(* IEC 61131-3 sources: repolevel_ST_code_completion/real_groud_truth最新/repoeval_open-type_dual-axis_winding_machine/readful_result, 5 files *)

(* ---- CheckF.st ---- *)
VAR
END_VAR

IF lM >= lL AND lM <= lH THEN
    lF := lM;
ELSE
    IF lM < lL THEN
        lF := lL;
    ELSE
        lF := lH;
    END_IF
END_IF

(* ---- F_CalculateRadius.st ---- *)
# --------------------------------------------------
# FUNCTION F_CalculateRadius : LREAL
# VAR_INPUT
# 	lD				:	LREAL;		//两轴中心距离
# 	lHold			:	LREAL;		//测量开始时的AxisV位置
# 	lHnew			:	LREAL;		//测量结束时的AxisV位置
# 	lTk				:	LREAL;		//材料厚度
# 	lOffset			:	LREAL;		//高度偏移量
# END_VAR
#
# // 计算从轴半径
# IF (lHnew - lHold) > 0.01 THEN  // 避免除零
# 	F_CalculateRadius := lD / 2 + (lHnew - lHold) / 2 + lTk + lOffset;
# ELSE
# 	F_CalculateRadius := lD / 2 + lTk + lOffset;
# END_IF
# --------------------------------------------------
# the below code fragment can be found in:
# 开放式双轴卷绕机编程开发实训-PRG\PLC_PRG.st
# --------------------------------------------------
# 			// 使用F_CalculateRadius函数计算从轴半径
# 			Sr := F_CalculateRadius(lD := AxisDistance, lHold := AxisVStart, lHnew := AxisVEnd, lTk := MaterialThickness, lOffset := HeightOffset);
#
# 			// 调用F_CompensateVelocity函数计算速度补偿
# 			CompensatedVelocity := F_CompensateVelocity(lCurrentVel := CurrentVelocity, lOldPos := OldPosition, lNewPos := NewPosition, lRadius := Sr, lTk := MaterialThickness, bUnwinding := IsUnwinding);

(* ---- F_CompensateVelocity.st ---- *)
// Velocity compensation formula:
// V_compensated = V_current * (R_old / R_new)

VAR
    lOldRadius : LREAL; // Previous radius
    lNewRadius : LREAL; // Current radius
END_VAR

// Calculate the old and new radii based on the positions and material thickness
lOldRadius := ABS(SQRT(EXPT(lRadius, 2) + EXPT(lOldPos, 2)) - SQRT(EXPT(lRadius, 2) + EXPT(lOldPos - lTk, 2))) / SMC_PI + lTk;
lNewRadius := ABS(SQRT(EXPT(lRadius, 2) + EXPT(lNewPos, 2)) - SQRT(EXPT(lRadius, 2) + EXPT(lNewPos - lTk, 2))) / SMC_PI + lTk;

// Adjust velocity based on unwinding or winding direction
IF bUnwinding THEN
    F_CompensateVelocity := lCurrentVel * (lOldRadius / lNewRadius);
ELSE
    F_CompensateVelocity := lCurrentVel * (lNewRadius / lOldRadius);
END_IF;

(* ---- SeekHome.st ---- *)
VAR
	_fbMoveVel	:	MC_MoveVelocity;
	_fbMoveAbs	:	MC_MoveAbsolute;
	_fbHalt		:	MC_Halt;
	_fbSetPos	:	MC_SetPosition;
	_fbRtrig		:	R_TRIG;
	_fbFtrig		:	F_TRIG;
	_nBDirection	:	MC_DIRECTION;
	_fTempPos		:	LREAL;
	_nState		:	USINT;
END_VAR

METHOD FAST_ZERO
VAR_IN_OUT
	_Axis	:	AXIS_REF_SM3;
END_VAR
VAR_INPUT
	_xHome	:	BOOL;
	_xAbort	:	BOOL;
	_nHomeMode	:	HomeMode;
	_fFastHomeVel	:	LREAL;
	_fSlowHomeVel	:	LREAL;
	_fHomeAcc		:	LREAL;
	_fHomeDec		:	LREAL;
	_fHomePos		:	LREAL;
	_xReferenceSwitch	:	BOOL;//typically is true
	_nDirection	:	MC_DIRECTION;
	_xIndexPulse	:	BOOL;
END_VAR
VAR_OUTPUT
	_xBusy	:	BOOL;
	_xDone	:	BOOL;
	_xErr	:	BOOL;
	_iErrId	:	DINT;
END_VAR
VAR
	_fbMoveVel	:	MC_MoveVelocity;
	_fbMoveAbs	:	MC_MoveAbsolute;
	_fbHalt		:	MC_Halt;
	_fbSetPos	:	MC_SetPosition;
	_fbRtrig		:	R_TRIG;
	_fbFtrig		:	F_TRIG;
	_nBDirection	:	MC_DIRECTION;
	_fTempPos		:	LREAL;
	_nState		:	USINT;
END_VAR

CASE _nState OF
	0: // Initialization
		_xBusy := TRUE;
		_xDone := FALSE;
		_xErr := FALSE;
		_iErrId := 0;
		_nState := 1;

	1: // Check Home Condition
		IF _xHome THEN
			_fbRtrig(CLK := _xHome);
			IF _fbRtrig.Q THEN
				_nState := 2;
			END_IF;
		END_IF;

	2: // Execute Fast Home Velocity
		_fbMoveVel(Axis := _Axis, Velocity := _fFastHomeVel, Acceleration := _fHomeAcc, Deceleration := _fHomeDec, Direction := _nDirection);
		IF _fbMoveVel.Done THEN
			_nState := 3;
		END_IF;

	3: // Execute Slow Home Velocity
		_fbMoveVel(Axis := _Axis, Velocity := _fSlowHomeVel, Acceleration := _fHomeAcc, Deceleration := _fHomeDec, Direction := _nDirection);
		IF _fbMoveVel.Done THEN
			_nState := 4;
		END_IF;

	4: // Set Position
		_fbSetPos(Axis := _Axis, Position := _fHomePos);
		IF _fbSetPos.Done THEN
			_nState := 5;
		END_IF;

	5: // Complete
		_xBusy := FALSE;
		_xDone := TRUE;
		_nState := 0;

ELSE
	_xErr := TRUE;
	_iErrId := -1; // Error ID
END_CASE;

(* ---- StaDisplay.st ---- *)
VAR
	_nState : USINT;
END_VAR

// Implementation of the StaDisplay function block
// This function block is used to display the status of the machine using output signals Y1 to Y6.
METHOD DisplayStatus : VOID
VAR_INPUT
	iStatus : INT; // Input status code
END_VAR
VAR_OUTPUT
	Y1, Y2, Y3, Y4, Y5, Y6 : BOOL; // Output signals representing different status indicators
END_VAR

// Reset all output signals to FALSE initially
Y1 := FALSE;
Y2 := FALSE;
Y3 := FALSE;
Y4 := FALSE;
Y5 := FALSE;
Y6 := FALSE;

// Set the corresponding output signal based on the input status code
CASE iStatus OF
	1: Y1 := TRUE; // Status 1 - Activate Y1
	2: Y2 := TRUE; // Status 2 - Activate Y2
	3: Y3 := TRUE; // Status 3 - Activate Y3
	4: Y4 := TRUE; // Status 4 - Activate Y4
	5: Y5 := TRUE; // Status 5 - Activate Y5
	6: Y6 := TRUE; // Status 6 - Activate Y6
	ELSE
		// If the status code is not recognized, keep all outputs FALSE
END_CASE;
